TYPE TcoTixonPickStep_Control_v_1_x_x EXTENDS TcoTixonGenericControl : 
STRUCT
    {attribute addProperty Name "<#Stepper valve#> - q7"}
    StepperValve : BOOL;
END_STRUCT
END_TYPE

(* stored: Version 1.1.0.1, ProductVersion 3.1.4024.12
   DUT TcoTixonPickStep_Control_v_1_x_x: Id {f7e0b219-a242-0146-3a74-d187ed005bcf} *)
